FUNCTION Convert_LWORD_TO_LREAL : Hresult
VAR_INPUT
	in : LWORD;
	out : REFERENCE TO LREAL;
END_VAR
VAR
	converted : LREAL;
END_VAR
VAR CONSTANT
	INCOMPATIBLE : HRESULT := 16#9811070E;
END_VAR

converted := LWORD_TO_LREAL(in);

IF (LREAL_TO_LWORD(converted) <> in) THEN
	Convert_LWORD_TO_LREAL := INCOMPATIBLE;
	RETURN;
END_IF

out := converted;

END_FUNCTION

(* stored: Version 1.1.0.1, ProductVersion 3.1.4024.12
   POU Convert_LWORD_TO_LREAL: Id {95078546-1799-4011-a815-4fa641f687a1}, SpecialFunc None *)
